// TIA Portal V18 export
DATA_BLOCK "PartData_Interface_DB"   // DB1500
{ S7_Optimized_Access := 'TRUE' }
VERSION : 0.1
// stored: AutoNumber true, DBAccessibleFromOPCUA true, DBAccessibleFromWebserver true, IsOnlyStoredInLoadMemory false, IsRetainMemResEnabled false, IsWriteProtectedInAS false, MemoryReserve 100
   VAR
      PartDataID : Int := 1;   // 物料数据序号
      PartData { S7_SetPoint := 'True'} : Array[1..4] of "PartData_UDT";
      PartCMD : Array[1..4] of Struct
         Set : Bool;
         Use : Bool;
      END_STRUCT;
   END_VAR
BEGIN
   // PartData[1] : XXX物料
   // PartData[2] : XXX物料
   // PartData[3] : XXX物料
   // PartData[4] : XXX物料
END_DATA_BLOCK
